PROGRAM MAIN
VAR
END_VAR

END_PROGRAM

(* stored: Version 1.1.0.1
   POU MAIN: Id {9d3e4a85-922f-4849-a3e7-0fb22dde0815} *)
